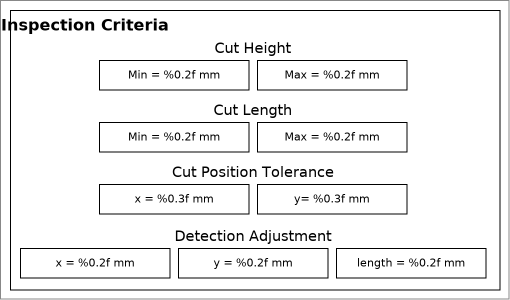
VISUALIZATION Settings_PassCriteria  // 510x300
VAR_IN_OUT
	CutHeightMin	: LREAL;
	CutHeightMax	: LREAL;
	CutLengthMin	: LREAL;
	CutLengthMax	: LREAL;
	CutToleranceX	: LREAL;
	CutToleranceY	: LREAL;
	AdjustmentX		: LREAL;
	AdjustmentY		: LREAL;
	AdjustmentLength: LREAL;
END_VAR
    Rectangle (10,10 490x280)
    Label (203,95 100x30), "Cut Length"
    Rectangle (99,122 150x30), "Min = %0.2f mm", text variable: CutLengthMin
        OnMouseClick: write CutLengthMin via Default
    Rectangle (257,122 150x30), "Max = %0.2f mm", text variable: CutLengthMax
        OnMouseClick: write CutLengthMax via Default, title 'Cut Position Y'
    Label (213,33 80x30), "Cut Height"
    Rectangle (99,60 150x30), "Min = %0.2f mm", text variable: CutHeightMin
        OnMouseClick: write CutHeightMin via Default
    Rectangle (257,60 150x30), "Max = %0.2f mm", text variable: CutHeightMax
        OnMouseClick: write CutHeightMax via Default, title 'Cut Position Y'
    Label (168,157 170x30), "Cut Position Tolerance"
    Rectangle (99,184 150x30), "x = %0.3f mm", text variable: CutToleranceX
        OnMouseClick: write CutToleranceX via Default
    Rectangle (257,184 150x30), "y= %0.3f mm", text variable: CutToleranceY
        OnMouseClick: write CutToleranceY via Default, title 'Cut Position Y'
    Label (173,221 160x30), "Detection Adjustment"
    Rectangle (20,248 150x30), "x = %0.2f mm", text variable: AdjustmentX
        OnMouseClick: write AdjustmentX via Default, title 'Cut Position X'
    Rectangle (178,248 150x30), "y = %0.2f mm", text variable: AdjustmentY
        OnMouseClick: write AdjustmentY via Default, title 'Cut Position Y'
    Rectangle (336,248 150x30), "length = %0.2f mm", text variable: AdjustmentLength
        OnMouseClick: write AdjustmentLength via Default, title 'Cut Position Y'
    Label (10,10 150x30), "Inspection Criteria"
END_VISUALIZATION

(* stored: Version 1.1.0.1, ProductVersion 3.1.4024.3
   Visu Settings_PassCriteria: Id {8f541173-aef9-4f48-902c-a4de07208827} *)
